PROGRAM MAIN
VAR
	
	test1: BOOL;
END_VAR

test1 := TRUE;

END_PROGRAM

(* stored: Version 1.1.0.1, ProductVersion 3.1.4024.11
   POU MAIN: Id {362ce905-19b7-4446-9237-c9ceaaf0217a}, SpecialFunc None *)
